VAR_OUTPUT
	qc : INT;
	//ActPOS : LREAL;
	//ActVelo : LREAL;
	//PosDiff : REAL;
	//exceptionMessage : STRING := '';
	BrakeEnabledCounter : DINT := 0;
	StaticCounter : DINT := 0; 
		OnUpLimit : UDINT;
	OnDownLimit : UDINT;
		SmodeTargetPos : LINT;  //target position for move
END_VAR

VAR
	RMT_DeadmanOFFCOunter : DINT;
//	checker : BOOL;
	ScalingInt : DINT;
	checkingReal : LINT;
//	checkingInt: DINT;  //only used for program
	
	//CurrentPosition : DINT;
	
	//SCALED VALUES FOR CALCULATIONS

	SmodeVel : LINT:= 10; //Maximum allowed velocity
	SmodeAcc : LINT:= 10; //Maximum allowed Acceleration
	SmodeDec : LINT:= 10;
	//SmodeJerk: ULINT:= 10; //Maximum change in Accel per loop
	SmodeWindow : LINT:= 2000; //Allowed window for move to be complete
	
	sendVel : LINT := 10;  //Actual velocity to send to EtherCAT card
	sendAcc: LINT := 10;  //Actual Acceleration to send to EtherCAT card
	sendDec: LINT := 10;


	
END_VAR

IF NOT joystickMotion.DeadManOut THEN
			KidAxis.PDecel := LREAL_TO_DINT(GVL_Index.Decel_For_DeadMan );
			KidAxis.pVelMax := 0;
			deadCounter := deadCOunter + 1;
ELSE
	GVL_Modes.nMotion_Command := 2;
	deadCounter := 0;
END_IF

IF  KidAxis.status.ready THEN
	ScalingInt := LREAL_TO_INT(1/ GVL_Motion.lrEncoder_ScalingNum);
ELSE
	RETURN;
END_IF

	SmodeTargetPos := F_LimitTarget(LREAL_TO_DINT(KidAxis.modeTargetPos));// * scalingInt;
	SmodeVel := ABS(KidAxis.modeVel);// * scalingInt;
	SmodeAcc := DINT_TO_LINT(KidAxis.modeAcc);//* scalingInt;
	SmodeDec := DINT_TO_LINT(KidAxis.modeAcc);
	

	SmodeWindow := KidAxis.modeWindow;//* scalingInt;
	
	
IF kidAxis.CheckIn.momControl AND NOT (joystickMotion.DeadManOut)  THEN

	IF GVL_INDEX.Direction_Flipped THEN
		SmodeTargetPos := F_LimitTarget(GVL_Index.Home_Offset - (GVL_DriveParameters.targetpos_FromMom * ScalingInt) );
	ELSE
		SmodeTargetPos := F_LimitTarget((GVL_DriveParameters.targetpos_FromMom * ScalingInt) + GVL_Index.Home_Offset);
	END_IF
	SmodeVel := GVL_DriveParameters.modeVel_FromMom;
	SmodeAcc := (GVL_DriveParameters.modeAccel_FromMom/3);
	SmodeDec := (GVL_DriveParameters.modeDecel_FromMom/3) + 5;
	//IF SmodeDec < SmodeAcc THEN smodeDec := smodeAcc; END_IF
//SmodeJerk:=  SmodeAcc/2;//* scalingInt;
END_IF

	IF (NOT kidAxis.CheckIn.momControl OR GVL_HMI.MomControl_Bypass) THEN
		IF joyStickMotion.DeadManOut THEN smodeVel := ABS(LREAL_TO_LINT(GVL_Motion.rHoist_SelectedVelocity)) + 5; END_IF
		IF joyStickMotion.DeadManOut  THEN smodeAcc := ABS(LREAL_TO_LINT(GVL_IO.rJoystick_Feedback * LINT_TO_LREAL(KidAxis.modeAcc) / 100)) + 20; END_IF;
		IF joyStickMotion.DeadManOut THEN smodeDec := sModeDec + 200; END_IF;
	END_IF

IF (kidAxis.CheckIn.momControl AND NOT kidAxis.CheckIn.Rmt_DeadManPressed) AND NOT GVL_HMI.MomControl_Bypass THEN
	KidAxis.PDecel := GVL_Index.Decel_For_DeadMan;
	KidAxis.pVelMax := 0;
	IF RMT_DeadmanOFFCOunter < 0  THEN 
		RMT_DeadmanOFFCOunter := 0;
	END_IF
	RMT_DeadmanOFFCOunter := RMT_DeadmanOFFCOunter + 1;
	
	IF RMT_DeadmanOFFCOunter < 200  THEN 
		RETURN;
	END_IF
END_IF

IF  (joystickMotion.DeadManOut OR (kidAxis.CheckIn.momControl AND kidAxis.CheckIn.Rmt_DeadManPressed)) THEN
 	//GVL_DriveParameters.controlWord:=15; //ENABLE DRIVE
	IF RMT_DeadmanOFFCOunter > 0  THEN 
		RMT_DeadmanOFFCOunter := 0;
	END_IF
	RMT_DeadmanOFFCOunter := RMT_DeadmanOFFCOunter - 1;
	
	GVL_Modes.bDrive_Enable := TRUE;
	KidAxis.pVelMax := 0;
	IF RMT_DeadmanOFFCOunter > -300  THEN 
		RETURN;
	END_IF
 ELSE
	 //GVL_DriveParameters.controlWord := 7; 
	 GVL_Modes.bDrive_Enable := FALSE;
END_IF

		checkingreal :=   ( ScalingInt * kidAxis.pVelDem * LREAL_TO_LINT(ABS(KidAxis.pVelDem)) )/ (  SmodeDec ) ; //Higher means more damping

		IF DINT_TO_LINT(KidAxis.actualPos) + checkingreal - SmodeTargetPos  > smodeWindow  THEN
			sendVel := -1 * ABS(SmodeVel);	
			SendAcc := smodeAcc;
		ELSIF KidAxis.actualPos + checkingreal - smodeTargetPos <= -1 * smodeWindow THEN
			sendVel :=  ABS(SmodeVel);
			SendAcc := smodeAcc;
		ELSE
				SendVel :=0;
		END_IF
		

				IF KidAxis.ActualVel = 0 THEN 	KidAxis.isbusy := FALSE; END_IF
			SendDec := smodeDec;	
IF (NOT joystickMotion.DeadManOut AND NOT kidAxis.CheckIn.momControl)
	OR (kidAxis.CheckIn.momControl AND  NOT kidAxis.CheckIn.Rmt_DeadManPressed) THEN
		//SendAcc := GVL_Speeds.QuickStop_Accel;
		SendDec := GVL_Index.Decel_For_DeadMan;
		SendVel := 0;
END_IF


	
				
IF KidAxis.pVelDem > -1 AND KidAxis.pVelDem < 1  THEN
	StaticCounter := StaticCounter + 1;
	ELSE
	StaticCounter := 0;
END_IF

IF StaticCounter< 0 THEN staticCounter  := 10000;  END_IF

OnUPLimit :=  BOOL_TO_USINT((NOT gvl_iNDEX.DIRECTION_FLIPPED AND ((Kidaxis.pVelDem > 0 OR SmodeTargetPos >= KidAxis.actualPos) AND  NOT (GVL_Safe_IO.bLimit_Hard_Up OR GVL_SAFE_IO.bHard_UP_Bypass_Enable)))
	OR (gvl_iNDEX.DIRECTION_FLIPPED AND ((Kidaxis.pVelDem < 0 OR SmodeTargetPos <= KidAxis.actualPos) AND  NOT (GVL_Safe_IO.bLimit_Hard_Up OR GVL_SAFE_IO.bHard_UP_Bypass_Enable)))) ;

OnDownLimit :=  BOOL_TO_USINT((gvl_iNDEX.DIRECTION_FLIPPED  AND ((Kidaxis.pVelDem > 0 OR SmodeTargetPos >= KidAxis.actualPos) AND  NOT (GVL_Safe_IO.bLimit_Hard_Down OR GVL_SAFE_IO.bHard_Down_Bypass_Enable)))
	OR (NOT GVL_Index.Direction_Flipped AND ((Kidaxis.pVelDem < 0 OR SmodeTargetPos <= KidAxis.actualPos) AND  NOT (GVL_Safe_IO.bLimit_Hard_down OR GVL_SAFE_IO.bHard_Down_Bypass_Enable))));
	
IF NOT kidAxis.CheckIn.momControl AND (OnUpLimit > 0  OR OnDownLimit > 0)   THEN 
	SendDec := DINT_TO_LINT(GVL_Index.Decel_For_DeadMan);
		SendVel := LINT_TO_INT(0);
		SendAcc :=0;
	//	OnUpLimit:=1;
	//	OnDownLimit:=1;
ELSE

	//	IF OnUpLimit=1 AND OnDOwnLimit = 1 THEN OnUpLimit := 0;  OnDownLimit :=0; END_IF
END_IF
KidAxis.PDecel := 10 + LINT_TO_DINT(sendDec * 6/5 );
		IF LINT_TO_DINT(SendAcc) > 20000 THEN SendAcc := 20000; END_IF
		
		IF GVL_Safe_IO.bRelease_Motor_Brake AND SendAcc <= 20000 THEN
			KidAxis.PAccel := LINT_TO_DINT(SendAcc);
				qc:= qc + 1;	
			KidAxis.pVelMax := LINT_TO_INT(SendVel);
			IF(ABS(SendVel)=1) THEN kidAxis.pVelMax := 0; END_IF
		
		END_IF
		

	//		Sendvel := 0;
	//ELSIF GVL_DriveParameters.actualpos - modePos + modewindow < (GVL_DriveParameters.actualVel *  GVL_DriveParameters.actualVel)/(1 + (2000 * modeAcc)) AND GVL_DriveParameters.actualVel>0 THEN
	//		Sendvel := 1;
	//ELSE
	//		sendVel := 2;
	//END_IF]]></ST>

ACTION MotionAtLimits:

END_ACTION

END_FUNCTION_BLOCK

// ---- POUs/Programs/Initialize/FB_FileCopy.TcPOU
FUNCTION_BLOCK FB_FileCopy
VAR_INPUT
        sSrcNetId                       : T_AmsNetId;(* TwinCAT network address of the source file *)
        sSrcPathName            : T_MaxString;(* Source file path and name *)
        sDestNetId              : T_AmsNetId;(* TwinCAT network address of the destination file *)
        sDestPathName           : T_MaxString; (* Destination file path and name *)
        bExecute                        : BOOL; (* Rising edge start fb execution *)
        tTimeOut                        : TIME := DEFAULT_ADS_TIMEOUT;(* Max. ADS timeout time *)
END_VAR
VAR_OUTPUT
        bBusy                   :BOOL;(* TRUE => File copy execution in progress, FALSE => File copy execution idle *)
 bError                  :BOOL;(* TRUE => Error, FALSE => No error *)
 nErrId                  :UDINT;(* Error code *)
END_VAR
VAR
        fbFileOpen              :FB_FileOpen;
        fbFileClose             :FB_FileClose;
        fbFileRead              :FB_FileRead;
        fbFileWrite             :FB_FileWrite;

        hSrcFile                        :UINT   := 0;(* File handle of the source file *)
 hDestFile                       :UINT   := 0;(* File handle of the destination file *)

        Step                    :DWORD;
        RisingEdge              :R_TRIG;

        buffRead                        :ARRAY[1..1000] OF BYTE;(* Buffer *)
 cbReadLength            :UDINT := 0;
END_VAR

RisingEdge(CLK:=bExecute);

CASE Step OF
        0:      (* Idle state *)
         IF RisingEdge.Q THEN
                        bBusy := TRUE;
                        bError:= FALSE;
                        nErrId:=0;
                        Step := 1;
                        cbReadLength:=0;
                        hSrcFile:=0;
                        hDestFile:=0;
                END_IF

        1:      (* Open source file *)
         fbFileOpen( bExecute := FALSE );
                fbFileOpen( sNetId := sSrcNetId, sPathName := sSrcPathName,
                        nMode := FOPEN_MODEREAD OR FOPEN_MODEBINARY,
                        ePath := PATH_GENERIC, tTimeout := tTimeOut, bExecute := TRUE );
                Step := Step + 1;
        2:
                fbFileOpen( bExecute := FALSE );
                IF NOT fbFileOpen.bBusy THEN
                        IF fbFileOpen.bError THEN
                                nErrId := fbFileOpen.nErrId;
                                bError := TRUE;
                                Step := 50;
                        ELSE
                                hSrcFile := fbFileOpen.hFile;
                                Step := Step + 1;
                        END_IF
                END_IF

        3:      (* Open destination file *)
         fbFileOpen( bExecute := FALSE );
                fbFileOpen( sNetId := sDestNetId, sPathName := sDestPathName,
                        nMode := FOPEN_MODEWRITE OR FOPEN_MODEBINARY,
                        ePath := PATH_GENERIC, tTimeout := tTimeOut, bExecute := TRUE );
                Step := Step+1;
        4:
                fbFileOpen( bExecute := FALSE );
                IF NOT fbFileOpen.bBusy THEN
                        IF fbFileOpen.bError THEN
                                nErrId := fbFileOpen.nErrId;
                                bError := TRUE;
                                Step := 50;
                        ELSE
                                hDestFile := fbFileOpen.hFile;
                                Step := Step + 1;
                        END_IF
                END_IF

        5:      (* Read data from source file *)
         cbReadLength := 0;
                fbFileRead( bExecute:= FALSE );
                fbFileRead( sNetId:=sSrcNetId, hFile:=hSrcFile,
                        pReadBuff:= ADR(buffRead), cbReadLen:= SIZEOF(buffRead),
                        bExecute:=TRUE, tTimeout:=tTimeOut );
                Step := Step + 1;
        6:
                fbFileRead( bExecute:= FALSE );
                IF NOT fbFileRead.bBusy THEN
                        IF fbFileRead.bError THEN
                                nErrId := fbFileRead.nErrId;
                                bError := TRUE;
                                Step := 50;
                        ELSE
                                cbReadLength := fbFileRead.cbRead;
                                Step := Step + 1;
                        END_IF
                END_IF

        7:      (* Write data to destination file *)
         fbFileWrite( bExecute := FALSE );
                fbFileWrite( sNetId:=sDestNetId, hFile:=hDestFile,
                        pWriteBuff:= ADR(buffRead), cbWriteLen:= cbReadLength,
                        bExecute:=TRUE, tTimeout:=tTimeOut );
                Step := Step + 1;
        8:
                fbFileWrite( bExecute := FALSE );
                IF NOT fbFileWrite.bBusy THEN
                        IF fbFileWrite.bError THEN
                                nErrId := fbFileWrite.nErrId;
                                bError := TRUE;
                                Step := 50;
                        ELSE
                                IF fbFileRead.bEOF THEN (* Check if the EOF flag ist set *)
                                 Step := 50;(* Cleanup: close the destination and source files *)
                         ELSE
                                        Step := 5; (* Repeat reading/writing *)
                         END_IF
                        END_IF
                END_IF

        30:     (* Close the destination file *)
         fbFileClose( bExecute := FALSE );
                fbFileClose( sNetId:=sDestNetId, hFile:=hDestFile, bExecute:=TRUE, tTimeout:=tTimeOut );
                Step := Step + 1;
        31:
                fbFileClose( bExecute := FALSE );
                IF NOT fbFileClose.bBusy THEN
                        IF fbFileClose.bError THEN
                                nErrId := fbFileClose.nErrId;
                                bError := TRUE;
                        END_IF
                        Step := 50;
                        hDestFile := 0;
                END_IF

        40: (* Close source file *)
         fbFileClose( bExecute := FALSE );
                fbFileClose( sNetId:=sSrcNetId, hFile:=hSrcFile, bExecute:=TRUE, tTimeout:=tTimeOut );
                Step := Step + 1;
        41:
                fbFileClose( bExecute := FALSE );
                IF NOT fbFileClose.bBusy THEN
                        IF fbFileClose.bError THEN
                                nErrId := fbFileClose.nErrId;
                                bError := TRUE;
                        END_IF
                        Step := 50;
                        hSrcFile := 0;
                END_IF

        50: (* Error or ready => Cleanup *)
         IF ( hDestFile <> 0 ) THEN
                        Step := 30; (* Close the destination file*)
         ELSIF (hSrcFile <> 0 ) THEN
                        Step := 40; (* Close the source file *)
         ELSE
                        Step := 0;      (* Ready *)
                        bBusy := FALSE;
                END_IF

END_CASE

END_FUNCTION_BLOCK

// ---- POUs/Programs/Main Program/EtherCATComs.TcPOU
PROGRAM EtherCATComs //Handles all comunication over ethercat on ParamUpdate Task
VAR
	//QuickUpdate : FB_CheckIn_EtherCAT;
	ParamUpdate : FB_EtherCATReader;
	ParameterID_FromMom AT %I* : USINT;
	ParameterID_ToMom AT %Q*: USINT;
END_VAR

//ParamUpdate();
//ParameterID_ToMom := ParamUpdate.ID;
ParamUpdate();

END_PROGRAM

// ---- POUs/Programs/P_AxisDataSelect.TcPOU
PROGRAM P_AxisDataSelect
VAR
	//bExternalControlEnable: BOOL;
	//CtrWord1: USINT;
	//CtrWord2: USINT;
END_VAR

//IF GVL_PLC.bMomTotalControl THEN

//CtrWord1 := UINT_TO_USINT(GVL_DriveParameters.controlWord MOD 256);
//CtrWord2 := UINT_TO_USINT(GVL_DriveParameters.controlWord / 256);

//IF bExternalControlEnable THEN
	//GVL_AxisIOData.nDataOut2Hardware := GVL_AxisIOData.nDataOut2ExternalNC;
	//GVL_AxisIOData.nCtrl1Hardware := GVL_AxisIOData.nCtrl1ExternalNC;
	//GVL_AxisIOData.nCtrl2Hardware := GVL_AxisIOData.nCtrl2ExternalNC;
	
	//GVL_AxisIOData.nDataOut2Hardware := GVL_AxisIOData.nDataOut2ExternalNC;
	//GVL_AxisIOData.nCtrl1Hardware := CtrWord1;
	//GVL_AxisIOData.nCtrl2Hardware := CtrWord2;
//ELSE
//	GVL_AxisIOData.nDataOut2Hardware := GVL_AxisIOData.nDataOut2LocalNC;
//	GVL_AxisIOData.nCtrl1Hardware := GVL_AxisIOData.nCtrl1LocalNC;
//	GVL_AxisIOData.nCtrl2Hardware := GVL_AxisIOData.nCtrl2LocalNC;	
//END_IF

//KidAxis.ParameterReader();

END_PROGRAM

// ---- POUs/Programs/Serial/P_LEDstatus.TcPOU
PROGRAM P_LEDstatus
VAR
	bErrorRecovery: BOOL;
	fbR_Trig: R_Trig;
	fbPulse: FB_Pulse;
END_VAR

fbR_Trig(CLK:=NOT GVL_PLC.bSafetyError);

fbPulse(bEnable:= TRUE, tTimeOn:= GVL_HMI.tPulseTime, tTimeOff:= GVL_HMI.tPulseTime, bPulse=> );

IF fbR_Trig.Q THEN
	GVL_Serial.nJoystickLED := 6;
END_IF

IF GVL_PLC.bLocalKeySwitchInput THEN
		GVL_Serial.nJoystickLED := 5;
END_IF

IF GVL_PLC.bSafetyError OR
	NOT GVL_Safe_IO.bES_Local_Status THEN
	GVL_Serial.nJoystickLED := 3;
	GVL_Serial.bDeadmanLED := FALSE;
	GVL_Serial.bZonLED := FALSE;
END_IF

END_PROGRAM

// ---- POUs/Programs/Serial/P_Serial.TcPOU
PROGRAM P_Serial
VAR
END_VAR

P_EL600x();
P_LEDstatus();
P_SerialRemote();
P_JoystickSetup();

END_PROGRAM

// ---- POUs/Programs/Test Programs/P_ParameterComm.TcPOU
PROGRAM P_ParameterComm
VAR
	fbMC_Power: MC_Power;
	fbMC_WriteParameter: MC_WriteParameter;
	bWrite: BOOL;
	fbMC_MoveAbsolute: MC_MoveAbsolute;
	fb_MC_MoveAbsolute: MC_MoveAbsolute;
END_VAR


//This function calls the ReadStatus of the axis.	
kidAxis.ReadStatus();


fbMC_Power(
	Axis:= kidAxis, 
	Enable:= GVL_Modes.bDrive_Enable, 
	Enable_Positive:= , 
	Enable_Negative:= , 
	Override:= GVL_Modes.lrDrive_Override, 
	BufferMode:= , 
	Options:= , 
	Status=> , 
	Busy=> , 
	Active=> , 
	Error=> , 
	ErrorID=> );
	



fbMC_WriteParameter(
	Axis:= kidaxis, 
	Execute:= bWrite, 
	ParameterNumber:= AxisEnPositionLagMonitoring, 
	Value:= 1, 
	Done=> , 
	Busy=> , 
	Error=> , 
	ErrorID=> );
	
fbMC_MoveAbsolute.Position := GVL_Index.Target_Down;
	
	
fbMC_MoveAbsolute(
	Axis:= kidAxis, 
	Execute:= bStart_Motion, 
	Position:= , 
	Velocity:= 360, 
	Acceleration:= , 
	Deceleration:= , 
	Jerk:= , 
	BufferMode:= , 
	Options:= , 
	Done=> , 
	Busy=> , 
	Active=> , 
	CommandAborted=> , 
	Error=> , 
	ErrorID=> );

ACTION A_MC_MoveAbsolute:




fb_MC_MoveAbsolute(
	Axis:= kidAxis, 
	Execute:= bStart_Motion, 
	Position:= 0, 
	Velocity:= , 
	Acceleration:= , 
	Deceleration:= , 
	Jerk:= , 
	BufferMode:= , 
	Options:= , 
	Done=> , 
	Busy=> , 
	Active=> , 
	CommandAborted=> , 
	Error=> , 
	ErrorID=> );
END_ACTION

END_PROGRAM
